PROGRAM pouS1Warnings
VAR
END_VAR

// NETWORK 1

END_PROGRAM

(* stored: Version 1.1.0.1, ProductVersion 3.1.4024.12
   POU pouS1Warnings: Id {65a0745a-e675-400f-ad40-91f4efb6ca28}, SpecialFunc None *)
